Staubli VAL3: Blend.pjx

--- Blend.pjx ---
Parameters version=s7.9 stackSize=5000 millimeterUnit=true
Program file=start.pgx
Program file=stop.pgx
Data file=Blend.dtx

--- JointBlend.pgx ---
program JointBlend()
begin
end
